{attribute 'qualified_only'}
{attribute 'strict'}
TYPE E_ErrorId :
(
	PASSIVE_ABORT := 16#FFFFFFFF
)UDINT;
END_TYPE

(* stored: Version 1.1.0.1, ProductVersion 3.1.4024.12
   DUT E_ErrorId: Id {83c8117b-addc-4864-8fd8-2c13fc05b90a} *)
